PROGRAM OP150_Lsr
VAR
	
END_VAR

END_PROGRAM

(* stored: Version 1.1.0.1, ProductVersion 3.1.4024.11
   POU OP150_Lsr: Id {41dcda6c-df8c-48f4-9604-24709f23232f}, SpecialFunc None *)
